FUNCTION ToSwTimestamp_Mode : BOOL
VAR_INPUT
	ipChObject : I_CH_OBJECT;
	ipSwTimestamp_Mode : REFERENCE TO I_SwTimestamp_Mode;
END_VAR

VAR
	ipTmp : I_SwTimestamp_Mode;
END_VAR

(* 
   1. Test if the interface exists
   2. Test if the object implements a "Object" interface 
   3. Write reference to interface in parameter
   4. Returne TRUE if succesfull
*)
IF ipChObject <> 0 AND_THEN __QUERYINTERFACE(ipChObject,ipTmp) THEN
	ipSwTimestamp_Mode := ipTmp;
	ToSwTimestamp_Mode := TRUE;
END_IF

END_FUNCTION

(* stored: Version 1.1.0.1, ProductVersion 3.1.4024.12
   POU ToSwTimestamp_Mode: Id {05bfc70d-4ab4-4686-89f6-c06716a045be}, SpecialFunc None *)
